FUNCTION_BLOCK Fail_scenarios (* Composite Function Block Type *)
  (* Standard: 61499-2 *)
  (* Version 0.0, 5/14/2019, erik, nxtControl GmbH, template *)
  PACKAGE Main;
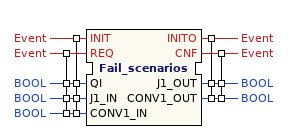
  EVENT_INPUT
    INIT WITH QI, J1_IN, CONV1_IN; (* Initialization Request *)
    REQ WITH QI, J1_IN, CONV1_IN; (* Normal Execution Request *)
  END_EVENT
  EVENT_OUTPUT
    INITO WITH J1_OUT, CONV1_OUT; (* Initialization Confirm *)
    CNF WITH J1_OUT, CONV1_OUT; (* Execution Confirmation *)
  END_EVENT
  VAR_INPUT
    QI : BOOL; (* Input event qualifier *)
    J1_IN : BOOL;
    CONV1_IN : BOOL;
  END_VAR
  VAR_OUTPUT
    J1_OUT : BOOL;
    CONV1_OUT : BOOL;
  END_VAR
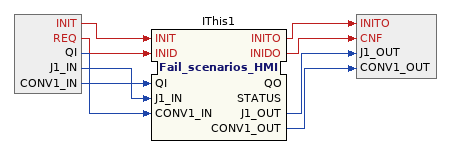
  FBS
    IThis1 : Fail_scenarios_HMI;
  END_FBS
  EVENT_CONNECTIONS
    INIT TO IThis1.INIT;
    REQ TO IThis1.INID;
    IThis1.INITO TO INITO;
    IThis1.INIDO TO CNF;
  END_CONNECTIONS
  DATA_CONNECTIONS
    QI TO IThis1.QI;
    J1_IN TO IThis1.J1_IN;
    CONV1_IN TO IThis1.CONV1_IN;
    IThis1.J1_OUT TO J1_OUT;
    IThis1.CONV1_OUT TO CONV1_OUT;
  END_CONNECTIONS
END_FUNCTION_BLOCK
